Yaskawa INFORM job: R1_72,2(0,0)KM-OK_MOD.JBI

/JOB
//NAME R1_72,2(0,0)KM-OK_MOD
///FOLDERNAME KRIS-SCIANA
//POS
///NPOS 95,95,0,4,0,0
///TOOL 0
///POSTYPE PULSE
///PULSE
C00000=214739,-34142,-86579,18171,90882,-33584
C00001=192628,-9219,-68940,27221,97535,-38774
C00002=192628,-9219,-68940,27221,97535,-38774
C00003=206785,1928,-2866,24835,77749,-31705
C00004=211412,-5691,-9151,24019,76339,-30254
C00005=211721,-3296,-4468,24119,74735,-30470
C00006=211721,-2988,-3159,24186,74143,-30595
C00007=211721,-3286,-4423,24121,74715,-30475
C00008=212044,-1475,-2934,24060,74632,-30369
C00009=211721,-3286,-4423,24121,74715,-30475
C00010=204612,2210,-14410,24827,85008,-30989
C00011=203386,32246,31282,35331,81776,-30118
C00012=203386,38484,48235,36062,75846,-32062
C00013=208339,32558,44817,36137,73023,-30932
C00014=209835,42985,55078,32968,75720,-29181
C00015=209835,44613,58630,33147,74579,-29524
C00016=208515,35726,50678,36597,71167,-31509
C00017=208862,38262,53326,36655,70758,-31505
C00018=208339,32558,44817,36137,73023,-30932
C00019=204483,35517,43983,35840,76221,-31482
C00020=204612,2210,-14410,24827,85008,-30989
C00021=204612,18022,-42675,26555,108188,-25943
C00022=214739,-34142,-86579,18171,90882,-33584
C00023=216406,-37850,-86218,17444,88554,-33440
C00024=217080,-39257,-86022,17157,87628,-33372
C00025=216891,-43789,-85751,17261,85277,-33761
C00026=217262,-41380,-84303,17098,85542,-33611
C00027=217436,-41971,-84662,17026,85428,-33572
C00028=217080,-39257,-86022,17157,87628,-33372
C00029=216120,-38690,-85533,17566,87791,-33633
C00030=216269,-39865,-84982,17508,86862,-33722
C00031=216120,-38690,-85533,17566,87791,-33633
C00032=217080,-39257,-86022,17157,87628,-33372
C00033=201345,-20375,-78021,31054,112530,-39584
C00034=201639,-23474,-77107,30489,110579,-40057
C00035=202590,-24455,-77954,30278,110316,-39807
C00036=201639,-23474,-77107,30489,110579,-40057
C00037=201345,-20375,-78021,31054,112530,-39584
C00038=205311,-24199,-81401,30131,111496,-38553
C00039=204414,-22055,-81146,30572,112570,-38540
C00040=202220,-16510,-80317,31730,115203,-38470
C00041=184984,-3292,-66527,21578,97839,-52041
C00042=187848,106335,29423,-5768,95800,74791
C00043=187846,93398,30248,-5715,88678,75115
C00044=187845,90841,31211,-5716,86781,75201
C00045=186749,80935,25217,37882,97144,45469
C00046=188249,88132,29282,-5868,86603,75331
C00047=187781,90810,31570,-5693,86541,75193
C00048=186593,79700,23961,37938,97314,45468
C00049=186285,79829,24181,38011,97380,45375
C00050=186155,80197,24595,38034,97381,45324
C00051=185994,80326,25273,38042,97165,45186
C00052=185838,79602,22632,38213,98224,45505
C00053=185327,80011,19037,38655,100344,46081
C00054=124459,133068,90612,6691,115644,64898
C00055=124459,133068,90612,6691,115644,64898
C00056=93275,113796,34371,-3502,120109,70620
C00057=89315,113601,52844,2619,120646,72485
C00058=89316,111310,53557,2572,119031,72446
C00059=89697,121055,69415,651,117839,72105
C00060=89348,111517,54075,2569,118818,72453
C00061=89564,113087,57614,2554,117442,72498
C00062=90033,119920,67876,706,118200,72231
C00063=91337,116538,63361,923,119232,72724
C00064=99842,93639,33750,-17614,115849,72169
C00065=99880,92745,32649,-17651,116064,72149
C00066=99324,86551,24395,-17976,117766,71666
C00067=94613,96171,29214,-8772,122473,71759
C00068=95513,127998,72000,-2391,121454,32503
C00069=95373,128312,72443,-2414,81128,32453
C00070=95373,169527,125925,-4488,33256,32455
C00071=126436,146554,76460,6599,53537,-23923
C00072=95373,169524,125926,-4503,33256,32457
C00073=142575,-91178,-115388,39866,103652,-54544
C00074=192628,-9219,-68940,27221,97535,-38774
C00075=206785,1928,-2866,24835,77749,-31705
C00076=209029,-3383,-7279,24450,77069,-31002
C00077=209515,-206,-2001,24513,75448,-31160
C00078=211191,3700,1031,21799,76737,-30315
C00079=215265,-130,-2171,21101,75678,-28996
C00080=214513,-2176,-4685,21195,76334,-29157
C00081=209029,-3383,-7279,24450,77069,-31002
C00082=204612,2210,-14410,24827,85008,-30989
C00083=203386,32246,31282,35331,81776,-30118
C00084=203386,38484,48235,36062,75846,-32062
C00085=206012,36095,48449,36242,73649,-31703
C00086=207229,41756,57711,36730,70874,-32148
C00087=210692,36139,51784,36533,70057,-30957
C00088=208339,32558,44817,36137,73023,-30932
C00089=204483,35517,43983,35840,76221,-31482
C00090=204612,2210,-14410,24827,85008,-30989
C00091=192628,-9219,-68940,27221,97535,-38774
C00092=135854,-98188,-118079,40471,104995,-56824
C00093=123760,23071,-66067,30293,113844,-22684
C00094=95373,169527,125925,-4488,33256,32455
BC00000=352013,15,1075175
BC00001=352013,15,1075175
BC00002=365574,15,642260
BC00003=365574,15,642260
BC00004=365574,15,642260
BC00005=365574,15,642260
BC00006=365574,15,642260
BC00007=365574,15,642260
BC00008=365574,15,642260
BC00009=365574,15,642260
BC00010=365574,15,642260
BC00011=365574,15,642260
BC00012=365574,15,642260
BC00013=365574,15,642260
BC00014=365574,15,642260
BC00015=365574,15,642260
BC00016=365574,15,642260
BC00017=365574,15,642260
BC00018=365574,15,642260
BC00019=365574,15,642260
BC00020=365574,15,642260
BC00021=365574,15,1075175
BC00022=352013,15,1075175
BC00023=346494,15,1075175
BC00024=344287,15,1075175
BC00025=341901,15,1075175
BC00026=341901,15,1075175
BC00027=344290,15,1075175
BC00028=344287,15,1075175
BC00029=338131,15,1075175
BC00030=338132,15,1075175
BC00031=338131,15,1075175
BC00032=344287,15,1075175
BC00033=302697,15,1075175
BC00034=302700,15,1075175
BC00035=302719,15,1075175
BC00036=302700,15,1075175
BC00037=302697,15,1075175
BC00038=316402,15,1075175
BC00039=317723,15,1075175
BC00040=321027,15,1075175
BC00041=333173,81717,1075175
BC00042=376146,194177,1075175
BC00043=376146,194177,1075175
BC00044=376277,192427,1075175
BC00045=398174,122098,1075175
BC00046=376329,191727,1075175
BC00047=376329,191727,1075175
BC00048=398174,122098,1075175
BC00049=398174,122098,1075175
BC00050=398174,122098,1075175
BC00051=398174,116514,1075175
BC00052=398174,116400,1075175
BC00053=398174,116114,1075175
BC00054=235371,182236,1075175
BC00055=16839,182236,1075175
BC00056=13012,209674,1075175
BC00057=13012,209674,1075175
BC00058=13735,213189,1075175
BC00059=14024,214595,1075175
BC00060=14024,214595,1075175
BC00061=14024,214595,1075175
BC00062=14024,214595,1075175
BC00063=14024,214595,1075175
BC00064=14024,214595,1075175
BC00065=14024,214595,1075175
BC00066=14024,214595,1075175
BC00067=14024,214595,1075175
BC00068=10344,234287,1075175
BC00069=10344,234287,1075175
BC00070=10345,234286,1075173
BC00071=262155,152897,1075174
BC00072=327786,234286,1075172
BC00073=352013,111996,1075175
BC00074=352013,15,1075175
BC00075=365574,15,642260
BC00076=365574,15,642260
BC00077=365574,15,642260
BC00078=365574,15,642260
BC00079=365574,15,642260
BC00080=365574,15,642260
BC00081=365574,15,642260
BC00082=365574,15,642260
BC00083=365574,15,642260
BC00084=365574,15,642260
BC00085=365574,15,642260
BC00086=365574,15,642260
BC00087=365573,15,642260
BC00088=365574,15,642260
BC00089=365574,15,642260
BC00090=365574,15,642260
BC00091=352013,15,1075175
BC00092=352013,397246,1075175
BC00093=249935,462030,1075174
BC00094=10345,614086,1075173
///POSTYPE BASE
///RECTAN
///RCONF 0,0,0,0,1,0,0,0,0,0,0,0,0,0,0,0,0,0,0,0,0,0,0,0
P00006=2.006,1.622,-0.565,0.0000,0.0000,0.0000
P00021=0.073,2.058,-0.109,0.0000,0.0000,0.0000
///RCONF 0,0,0,0,0,0,0,0,0,0,0,0,0,0,0,0,0,0,0,0,0,0,0,0
P00030=-0.014,-0.768,0.131,0.0000,0.0000,0.0000
P00031=-0.170,0.039,-0.647,0.0000,0.0000,0.0000
//INST
///DATE 2025/04/29 11:03
///ATTR SC,RW
///GROUP1 RB1,BS1
NOP
'R1_72.2(0,0)
'Path S1563
SFTOF
MOVJ C00000 BC00000 VJ=70.00
MOVJ C00001 BC00001 VJ=70.00
MOVJ C00002 BC00002 VJ=70.00
MOVJ C00003 BC00003 VJ=70.00
MOVL C00004 BC00004 V=166.7
MOVL C00005 BC00005 V=100.0
REFP 3 C00006 BC00006
CALL JOB:SEARCH-R1
SET P030 P006
SFTON P030
MOVL C00007 BC00007 V=100.0
REFP 3 C00008 BC00008
CALL JOB:SEARCH-R1
SET P030 P006
SFTON P030
MOVL C00009 BC00009 V=100.0
SFTOF
MOVL C00010 BC00010 V=400.0
MOVL C00011 BC00011 V=166.7
MOVL C00012 BC00012 V=166.7
MOVL C00013 BC00013 V=166.7
MOVL C00014 BC00014 V=100.0
REFP 3 C00015 BC00015
CALL JOB:SEARCH-R1
SET P031 P006
SFTON P031
MOVL C00016 BC00016 V=100.0
REFP 3 C00017 BC00017
CALL JOB:SEARCH-R1
SET P031 P006
SFTON P031
MOVL C00018 BC00018 V=100.0
SFTOF
MOVL C00019 BC00019 V=166.7
MOVL C00020 BC00020 V=400.0
MOVL C00021 BC00021 V=1000.0
MOVJ C00022 BC00022 VJ=70.00
MOVJ C00023 BC00023 VJ=50.00
MOVL C00024 BC00024 V=100.0
MOVL C00025 BC00025 V=60.0
REFP 3 C00026 BC00026
CALL JOB:SEARCH-R1
SET P021 P006
SFTON P021
MOVL C00027 BC00027 V=60.0
MOVL C00028 BC00028 V=100.0
MOVL C00029 BC00029 V=60.0
REFP 3 C00030 BC00030
CALL JOB:SEARCH-R1
SET P021 P006
SFTON P021
MOVL C00031 BC00031 V=60.0
MOVL C00032 BC00032 V=100.0
MOVL C00033 BC00033 V=100.0
MOVL C00034 BC00034 V=60.0
REFP 3 C00035 BC00035
CALL JOB:SEARCH-R1
SET P021 P006
SFTON P021
MOVL C00036 BC00036 V=60.0
MOVL C00037 BC00037 V=100.0
MOVL C00038 BC00038 V=100.0
MOVL C00039 BC00039 V=166.7
MOVL C00040 BC00040 V=166.7
'Path VIA1564
SFTOF
MOVJ C00041 BC00041 VJ=50.00
'Path W1561
SFTOF
SFTON P021
CALL JOB:COFNIJ_DRUT
MOVJ C00042 BC00042 VJ=50.00
MOVJ C00043 BC00043 VJ=100.00
MOVJ C00044 BC00044 VJ=100.00
MOVL C00045 BC00045 V=166.7 PL=0
REFP 1 C00046 BC00046
REFP 2 C00047 BC00047
MACRO1 MJ#(0) ARGF6
ARCON
MOVL C00048 BC00048 V=10.8
MOVL C00049 BC00049 V=10.8
MOVL C00050 BC00050 V=10.8
MOVL C00051 BC00051 V=10.8
ARCOF
MOVL C00052 BC00052 V=100.0
MOVL C00053 BC00053 V=166.7
SFTOF
'Path VIA1565
SFTOF
MOVJ C00054 BC00054 VJ=50.00
MOVJ C00055 BC00055 VJ=50.00
'Path W1566
SFTOF
SFTON P021
MOVJ C00056 BC00056 VJ=100.00
MOVJ C00057 BC00057 VJ=100.00
MOVJ C00058 BC00058 VJ=50.00
MOVL C00059 BC00059 V=100.0 PL=0
REFP 1 C00060 BC00060
REFP 2 C00061 BC00061
MACRO1 MJ#(0) ARGF5
ARCON
MOVL C00062 BC00062 V=8.3
MOVL C00063 BC00063 V=8.3
ARCOF
MOVL C00064 BC00064 V=10.0
ARCON
MOVL C00065 BC00065 V=8.3
MOVL C00066 BC00066 V=8.3
ARCOF
MOVL C00067 BC00067 V=166.7
MOVL C00068 BC00068 V=166.7
SFTOF
MOVJ C00069 BC00069 VJ=50.00
MOVJ C00070 BC00070 VJ=100.00
MOVJ C00071 BC00071 VJ=70.00
MOVL C00072 BC00072 V=1000.0
MOVJ C00073 BC00073 VJ=70.00
MOVJ C00074 BC00074 VJ=70.00
MOVJ C00075 BC00075 VJ=70.00
MOVL C00076 BC00076 V=166.7
SFTON P030
MOVL C00077 BC00077 V=100.0
MOVL C00078 BC00078 V=100.0 PL=0
MACRO1 MJ#(0) ARGF7
ARCON
MOVL C00079 BC00079 V=9.2
ARCOF
MOVL C00080 BC00080 V=233.3
SFTOF
MOVL C00081 BC00081 V=333.3
MOVL C00082 BC00082 V=400.0
MOVL C00083 BC00083 V=166.7
MOVL C00084 BC00084 V=166.7
MOVL C00085 BC00085 V=166.7
MACRO1 MJ#(0) ARGF6
SFTON P031
MOVL C00086 BC00086 V=166.7 PL=0
ARCON
MOVL C00087 BC00087 V=11.7
ARCOF
MOVL C00088 BC00088 V=100.0
SFTOF
MOVL C00089 BC00089 V=166.7
MOVL C00090 BC00090 V=400.0
MOVL C00091 BC00091 V=666.7
MOVJ C00092 BC00092 VJ=70.00
MOVJ C00093 BC00093 VJ=70.00
MOVJ C00094 BC00094 VJ=100.00
END
